// SIMATIC S7-200 SMART project (STEP 7-Micro/WIN SMART), CPU SR60

SYMBOL_TABLE 表格 3
夹爪正转i            V0.1
夹爪升i             V0.2
夹爪反转i            V0.3
夹爪退i             V0.4
夹爪停i             V0.5
夹爪进i             V0.6
夹爪紧i             V0.7
夹爪降i             V1.0
夹爪松i             V1.1
END_SYMBOL_TABLE

ORGANIZATION_BLOCK MAIN:OB1
TITLE=PLC
BEGIN
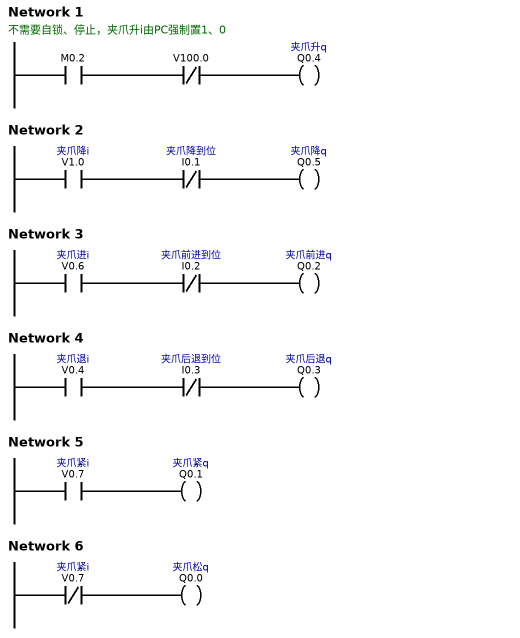
Network 1
// 不需要自锁、停止，夹爪升i由PC强制置1、0
LD     M0.2
AN     V100.0
=      夹爪升q:Q0.4
Network 2
LD     夹爪降i:V1.0
AN     夹爪降到位:I0.1
=      夹爪降q:Q0.5
Network 3
LD     夹爪进i:V0.6
AN     夹爪前进到位:I0.2
=      夹爪前进q:Q0.2
Network 4
LD     夹爪退i:V0.4
AN     夹爪后退到位:I0.3
=      夹爪后退q:Q0.3
Network 5
LD     夹爪紧i:V0.7
=      夹爪紧q:Q0.1
Network 6
LDN    夹爪紧i:V0.7
=      夹爪松q:Q0.0
END_ORGANIZATION_BLOCK
